        |   # first, check whether the corner is too low to the ground that the bottom homing will hit the ground (z < -400)
        |   lc_height = get_lift_column_height_condensed()
        |   # total height = zeroed lift column height (41.25 inches) (1.04775 m) plus lift column height plus robot relative height
        |   totalheight = 1.04775 + lc_height + point0[2]
        |   if totalheight < 1.04775 - 0.400:
        |     # bad
        |     popuptext = "Tank Corner is too low to the ground. Collisions will occur. Stop Program and raise tank. "
        |     # infinite loop
        |     while 1==1:
        |       popup(popuptext, title="Robot Positioning Warning",blocking=True)
        |     end
        |   end
        | 
        | 
        | 
        |   # next, check whether the touchpoints are reachable
        |   allvalid = check_structofpoints_validity(struct_touchpoints)
        |   if not allvalid:
        | 
        |     # then unreachable
        |     # generate message
        |     listproblems = ""
        |     listnames = ["ph1", "ph2", "ph3", "ph4", "ph5", "ph6", "ph7", "ph2up", "ph4up"]
        |     i = 0
        |     structlength = 9
        |     while i < structlength:
        |       curr = struct_touchpoints[i]
        |       valid = get_inverse_kin_has_solution(curr)
        |       if not valid:
        |         listproblems = listproblems + listnames[i]
        |       end
        |       i = i + 1
        |     end
        |     # display
        |     popuptext = "Robot is too far from tank corner. Cannot reach some necessary positions. Stop Program and move robot closer. " + listproblems
        |     # infinite loop
        |     while 1==1:
        |       popup(popuptext, title="Robot Positioning Warning",blocking=True)
        |     end
        |   end
        | 
        | end
        | 
        | # this function takes a struct of points as an argument, and checks whether every point in the list is reachable using get_inverse_kin_has_solution()
        | # this function does NOT check for weird twists or joint limits
        | # inputstruct must contain only points
        | # it returns true if all points are valid. it returns false if any points are valid
        | # a list of length 0 indicates that all points are valid
        | def check_structofpoints_validity(inputstruct):
        |   # next, check whether the touchpoints are reachable
        |   structlength = length(inputstruct)
        |   i = 0
        |   allvalid = True
        |   while i < structlength:
        |     curr = inputstruct[i]
        |     valid = get_inverse_kin_has_solution(curr)
        |     if not valid:
        |       return False
        |     end
        |     i = i + 1
        |   end
        |   return True
        | end
        | 
        | # checks the validity of all points during a left weld
        | # takes 2 arguments: struct1 (struct1[0] has to contain pointintersect) and struct2 (contains all the points (9) of the weld path)
        | def check_validity_left(struct1, struct2):
        |   #first, check whether robot is too close
        |   pointintersect = struct1[0]
        |   # next, check if the corner is too close to the robot to do a left around weld (complex but approximately X > -1300)
        |   # if y < 0, then x < -1300. if y < 480, then y > (1300+x)*8. if y > 480, then y > (1235+x)*4 + 500
        |   toocloseleftweld = False
        |   if pointintersect[1] < 0:
        |     if pointintersect[0] > -1.300:
        |       toocloseleftweld = True
        |     end
        |   elif pointintersect[1] < 0.480:
        |     if pointintersect[1] < (1.300 + pointintersect[0])*8:
        |       toocloseleftweld = True
        |     end
        |   else:
        |     if pointintersect[1] < (1.235 + pointintersect[0])*4 + 0.500:
        |       toocloseleftweld = True
        |     end
        |   end
        |   if toocloseleftweld:
        |     # bad
        |     popuptext = "Robot is too close to tank corner. Collisions may occur. Stop Program and move robot farther. "
        |     # infinite loop
        |     while 1==1:
        |       popup(popuptext, title="Robot Positioning Warning",blocking=True)
        |     end
        |   end
        | 
        |   #next, check whether all the points in the weldpath are valid
        |   structlength = 9
        |   i = 0
        |   allvalid = True
        |   listproblems = ""
        |   listnames = ["point1", "point2", "point4", "point5", "point_1", "point_2", "point_3", "point_4", "point_5"]
        |   while i < structlength:
        |     curr = struct2[i]
        |     valid = get_inverse_kin_has_solution(curr)
        |     if not valid:
        |       allvalid = False
        |       listproblems = listproblems + listnames[i]
        |     end
        |     i = i + 1
        |   end
        | 
        |   if not allvalid:
        |     # display
        |     popuptext = "Robot is too far from tank corner. Cannot reach some necessary positions. Stop Program and move robot closer. " + listproblems
        |     # infinite loop
        |     while 1==1:
        |       popup(popuptext, title="Robot Positioning Warning",blocking=True)
        |     end
        |   end
        | 
        |   # check whether the path involves weird turns or joint limits. currently just checks the first position
        |   p_prev = [-0.021118, -1.26292, 2.43578, 5.07088, -2.29912, 1.53362] #last point of left weld prerotate
        |   joints_1 = get_inverse_kin(struct2[0], p_prev) # struct2[0] is point1
        |   allGood = True
        |   i = 0
        |   structlength = 6
        |   while i < structlength:
        |     joint_curr = joints_1[i]
        |     # check for anything that exceeds joint limits
        |     degreesmax = 360 * pi / 180
        |     if joint_curr > degreesmax or joint_curr < degreesmax * -1:
        |       allGood = False
        |     end
        |     # check for anything that is significantly different than the aligned approach. could indicate a twist is needed. we dont want that
        |     maxdifference = 150 * pi / 180
        |     difference = joint_curr - p_prev[i]
        |     if difference > maxdifference or difference * -1 > maxdifference:
        |       allGood = False
        |     end
        |     i = i + 1
        |   end
        | 
        |   if not allGood:
        |     # call lift column extend function
        |     struct2 = floor_corner_lift_column_extend_left(struct2)
        | 
        |   end
        | 
        |   # return struct2 back
        |   return struct2
        | end
        | 
        | # checks the validity of all points during a right weld
        | def check_validity_right(struct1, struct2):
        |   # first, check whether the right pivot will bonk itself
        |   pointintersect = struct1[0]
        |   heading1 = struct1[1] # this is the direction that the welder will face when doing the right side of the box
        | 
        |   #first, check whether the heading is just too far offset
        |   # more than 15 degrees off of 45 is too much
        |   # normal heading is 216 degrees
        |   #201 degrees to 231 degrees
        |   heading1degrees = heading1 * 180 / pi
        |   if heading1degrees < 201 or heading1degrees > 231 :
        |     # then out of range
        |     popuptext = "Robot is not aligned at a 45 degree angle of corner (15 degree leeway). Collisions may occur. Stop Program and align robot. heading1degrees=" + str_cat("",heading1degrees)
        |     # infinite loop
        |     while 1==1:
        |       popup(popuptext, title="Robot Positioning Warning",blocking=True)
        |     end
        |   end
        | 
        |   #TODO: add the checks for whether x is too close, given the heading
        |   # add checks for whether x is too close, given the heading
        |   # different equations for whether heading offset > 5 degrees or less (inc. negative)
        |   headingoffset = heading1degrees - 216
        |   if headingoffset < 5:
        |     # then calculate a and b
        |     a = 0.4584 + -0.02369 * headingoffset
        |     b = (-1151.4 + 13.83 * headingoffset) / 1000
        |     # check whether x > a*y+b
        |     if pointintersect[0] > a * pointintersect[1] + b:
        |       # bad
        |       popuptext = "Robot is too close to tank corner or not at the right angle. Collisions may occur. Stop Program and align robot. "
        |       # infinite loop
        |       while 1==1:
        |         popup(popuptext, title="Robot Positioning Warning",blocking=True)
        |       end
        |     end
        |   else:
        |     # headingoffset > 5 degrees
        |     if pointintersect[1] < 0:
        |       if pointintersect[0] > -1150.0 / 1000.0:
        |         #bad
        |         popuptext = "Robot is too close to tank corner. Collisions may occur. Stop Program and align robot. "
        |         # infinite loop
        |         while 1==1:
        |           popup(popuptext, title="Robot Positioning Warning",blocking=True)
        |         end
        |       end
        |     else:
        |       # if x > .7736 y - 1101.9 then bad
        |       if pointintersect[0] > 0.7736 * pointintersect[1] - 1101.9 / 1000:
        |         popuptext = "Robot is too close to tank corner. Collisions may occur. Stop Program and align robot. "
        |         # infinite loop
        |         while 1==1:
        |           popup(popuptext, title="Robot Positioning Warning",blocking=True)
        |         end
        |       end
        |     end
        |   end
        | 
        |   #next, check whether all the points in the weldpath are valid
        |   structlength = 9
        |   i = 0
        |   allvalid = True
        |   listproblems = ""
        |   listnames = ["point1", "point2", "point4", "point5", "point_1", "point_2", "point_3", "point_4", "point_5"]
        |   while i < structlength:
        |     curr = struct2[i]
        |     valid = get_inverse_kin_has_solution(curr)
        |     if not valid:
        |       allvalid = False
        |       listproblems = listproblems + listnames[i]
        |     end
        |     i = i + 1
        |   end
        | 
        |   if not allvalid:
        |     # display
        |     popuptext = "Robot is too far from tank corner. Cannot reach some necessary positions. Stop Program and move robot closer. " + listproblems
        |     # infinite loop
        |     while 1==1:
        |       popup(popuptext, title="Robot Positioning Warning",blocking=True)
        |     end
        |   end
        | 
        |   # check whether the path involves weird turns or joint limits. currently just checks the first position
        |   p_prev = [-1.13307, -1.48911, 2.84785, 4.92357, -4.89059, 1.57184] #last point of right weld prerotate
        |   joints_1 = get_inverse_kin(struct2[0], p_prev) # struct2[0] is point1
        |   allGood = True
        |   i = 0
        |   structlength = 6
        |   while i < structlength:
        |     joint_curr = joints_1[i]
        |     # check for anything that exceeds joint limits
        |     degreesmax = 360 * pi / 180
        |     if joint_curr > degreesmax or joint_curr < degreesmax * -1:
        |       allGood = False
        |     end
        |     # check for anything that is significantly different than the aligned approach. could indicate a twist is needed. we dont want that
        |     maxdifference = 150 * pi / 180
        |     difference = joint_curr - p_prev[i]
        |     if difference > maxdifference or difference * -1 > maxdifference:
        |       allGood = False
        |     end
        |     i = i + 1
        |   end
        | 
        |   if not allGood:
        |     struct2 = floor_corner_lift_column_extend_right(struct2)
        |   end
        | 
        |   # return struct2 back
        |   return struct2
        | end
        | 
        | def floor_corner_lift_column_extend_right(struct2):
        |   # we know that p1 cannot be accessed without a twist
        |   # calculate the height needed to get to p1
        |   liftcolumnincrement = 2.0 # mm
        |   enoughHeightAdded = False
        |   liftColumnHeightTest = 0
        |   while not enoughHeightAdded:
        |     liftColumnHeightTest = liftColumnHeightTest + liftcolumnincrement
        |     # set the orig_joints for p1. p1 demo was joint angles of [-0.45, -31.79, 56.47, 333.06, -130.98, 87.87] (degrees)
        |     # which equals [-0.007853981633974475, -0.5548401692089968, 0.985587428601197, 5.812993606692308, -2.28603225426217, 1.5336208137274159]
        |     orig_joints = [-0.007853981633974475, -0.5548401692089968, 0.985587428601197, 5.812993606692308, -2.28603225426217, 1.5336208137274159]
        |     # get the modified point:
        |     origp1 = struct2[0]
        |     testp1 = p[origp1[0], origp1[1], origp1[2] - liftColumnHeightTest / 1000.0, origp1[3], origp1[4], origp1[5]]
        |     testpa1 = p[origp1[0]+0.05, origp1[1]+0.05, origp1[2] - liftColumnHeightTest / 1000, origp1[3], origp1[4], origp1[5]]
        |     enoughHeightAdded = can_pose_be_reached_without_twist(testp1, orig_joints) and can_pose_be_reached_without_twist(testpa1, orig_joints)
        |   end
        | 
        |   origp2 = struct2[1]
        |   testp2 = p[origp2[0], origp2[1], origp2[2] - liftColumnHeightTest / 1000.0, origp2[3], origp2[4], origp2[5]]
        |   origp4 = struct2[2]
        |   testp4 = p[origp4[0], origp4[1], origp4[2] - liftColumnHeightTest / 1000, origp4[3], origp4[4], origp4[5]]
        |   origp5 = struct2[3]
        |   testp5 = p[origp5[0], origp5[1], origp5[2] - liftColumnHeightTest / 1000, origp5[3], origp5[4], origp5[5]]
        | 
        | 
        | 
        |   liftcolumnzneeded = liftColumnHeightTest
        |   ret = struct(point1=testp1,point2=testp2,point4=testp4,point5=testp5,point_1=struct2[4],point_2=struct2[5],point_3=struct2[6],point_4=struct2[7],point_5=struct2[8])
        |   return ret
        | 
        | end
        | 
        | # this function gets called if you are doing a left floor corner extended, and the top is too high to reach (twists, etc.)
        | # this function takes the struct2 of weld points and modifies them (by subtracting from z) until the first weld point is reachable.
        | # it determines the height that the lift column needs to raise to make the first point reachable
        | # it then checks whether that height will allow the other points to be reachable
        | # if its all good, it sets the global variable liftcolumnzneeded, modifies struct2's points, and returns struct2
        | # if its not all good, then it displays an error message popup.
        | def floor_corner_lift_column_extend_left(struct2):
        |   # we know that p1 cannot be accessed without a twist
        |   # calculate the height needed to get to p1
        |   liftcolumnincrement = 2 # mm
        |   enoughHeightAdded = False
        |   liftColumnHeightTest = 0
        |   while not enoughHeightAdded:
        |     liftColumnHeightTest = liftColumnHeightTest + liftcolumnincrement
        |     # set the orig_joints for p1. p1 demo was joint angles of [-0.45, -31.79, 56.47, 333.06, -130.98, 87.87] (degrees)
        |     # which equals [-0.007853981633974475, -0.5548401692089968, 0.985587428601197, 5.812993606692308, -2.28603225426217, 1.5336208137274159]
        |     orig_joints = [-0.007853981633974475, -0.5548401692089968, 0.985587428601197, 5.812993606692308, -2.28603225426217, 1.5336208137274159]
        |     # get the modified point:
        |     origp1 = struct2[0]
        |     testp1 = p[origp1[0], origp1[1], origp1[2] - liftColumnHeightTest / 1000, origp1[3], origp1[4], origp1[5]]
        |     enoughHeightAdded = can_pose_be_reached_without_twist(testp1, orig_joints)
        |   end
        | 
        |   # check whether the other 3 points are valid
        |   valid = True
        |   # get the modified point
        |   origp2 = struct2[1]
        |   testp2 = p[origp2[0], origp2[1], origp2[2] - liftColumnHeightTest / 1000, origp2[3], origp2[4], origp2[5]]
        |   # p2 demo was joint angles of [-0.45, -21.2, 56.98, 321.95, -130.97, 87.85] (degrees)
        |   # which equals [-0.007853981633974475, -0.3700098014227975, 0.9944886077863679, 5.619087526795738, -2.285857721336971, 1.5332717478770168]
        |   orig_joints = [-0.007853981633974475, -0.3700098014227975, 0.9944886077863679, 5.619087526795738, -2.285857721336971, 1.5332717478770168]
        |   valid = valid and can_pose_be_reached_without_twist(testp2, orig_joints)
        |   # get the modified point
        |   origp4 = struct2[2]
        |   testp4 = p[origp4[0], origp4[1], origp4[2] - liftColumnHeightTest / 1000, origp4[3], origp4[4], origp4[5]]
        |   # p4 demo was joint angles of [-8.62, -43.23, 99.53, 213.86, -89.19, 40.78] (degrees)
        |   # which equals [-0.15044738152191103, -0.7545058356371478, 1.7371262045099545, 3.7325611383150696, -1.556659159853741, 0.7117452689632868]
        |   orig_joints = [-0.15044738152191103, -0.7545058356371478, 1.7371262045099545, 3.7325611383150696, -1.556659159853741, 0.7117452689632868]
        |   valid = valid and can_pose_be_reached_without_twist(testp4, orig_joints)
        |   # get the modified point
        |   origp5 = struct2[3]
        |   testp5 = p[origp5[0], origp5[1], origp5[2] - liftColumnHeightTest / 1000, origp5[3], origp5[4], origp5[5]]
        |   # p5 demo was joint angles of [-0.59, -34.36, 77.71, 226.7, -89.18, 48.81] (degrees)
        |   # which equals [-0.010297442586766533, -0.5996951309852511, 1.356295361724792, 3.9566614142711405, -1.5564846269285415, 0.8518952078984314]
        |   orig_joints = [-0.010297442586766533, -0.5996951309852511, 1.356295361724792, 3.9566614142711405, -1.5564846269285415, 0.8518952078984314]
        |   valid = valid and can_pose_be_reached_without_twist(testp5, orig_joints)
        | 
        |   if not valid:
        |     # display
        |     popuptext = "Top of Weld is too high above robot. Cannot reach some necessary positions. Stop Program and try again with a lower top point. "
        |     # infinite loop
        |     while 1==1:
        |       popup(popuptext, title="Robot Positioning Warning",blocking=True)
        |     end
        |   else:
        |     liftcolumnzneeded = liftColumnHeightTest
        |     ret = struct(point1=testp1,point2=testp2,point4=testp4,point5=testp5,point_1=struct2[4],point_2=struct2[5],point_3=struct2[6],point_4=struct2[7],point_5=struct2[8])
        |     return ret
        |   end
        | end
        | 
        | # this function calculates whether a given pose can be reached, and if it can, whether it requires a wrist twist (from the seed joint angles)
        | # arguments are target pose (p[x,y,z,rx,ry,rz]) and orig_joints which is the 6 joint angles of a pose that is close by the target pose and has the desired joint angles
        | # returns true if the pose is valid and requires no twist. If pose is valid but requires a twist, returns false. If pose is invalid, returns false.
        | def can_pose_be_reached_without_twist(pose, orig_joints):
        |   # first, determine if the pose is valid
        |   valid = get_inverse_kin_has_solution(pose)
        |   if not valid:
        |     return False
        |   end
        |   joints_1 = get_inverse_kin(pose, orig_joints)
        |   #iterate through the 6 joints
        |   allGood = True
        |   i = 0
        |   structlength = 6
        |   while i < structlength:
        |     joint_curr = joints_1[i]
        |     # check for anything that exceeds joint limits
        |     degreesmax = 360 * pi / 180
        |     if joint_curr > degreesmax or joint_curr < degreesmax * -1:
        |       allGood = False
        |     end
        |     # check for anything that is significantly different than the aligned approach. could indicate a twist is needed. we dont want that
        |     maxdifference = 150 * pi / 180
        |     difference = joint_curr - orig_joints[i]
        |     if difference > maxdifference or difference * -1 > maxdifference:
        |       allGood = False
        |     end
        |     i = i + 1
        |   end
        |   return allGood
        | end
        | 
        | # this function sends a signal to turn extrusion on
        | def turn_extrusion_on():
        |   # flush the channel
        |   resp0 = send_serial_signal(["u", "r", "?"])
        |   # send the signal
        |   resp1 = send_serial_signal(["u", "R", "1"])
        |   # if resp <> "uR1"
        |   if resp1 != [252,82,49]:
        |     # turn off extrusion and heating. inform calvin
        |     resp2 = send_serial_signal(["u", "R", "0"])
        |     resp3 = send_serial_signal(["u", "H", "0"])
        |     popuptext = "Error code encountered while trying to start extrusion. Find Calvin. "
        |     while 1==1:
        |       popup(popuptext, title="Extrusion Error Code",blocking=True)
        |       popup(resp1, blocking=True)
        |     end
        |   end
        | end
        | 
        | # this function sends a signal and receives a response
        | # signal is a list of 3 strings, 1 character each. first is u. second is the next character. third is final character
        | def send_serial_signal(signal):
        |   signal2char = signal[1]
        |   signal3char = signal[2]
        |   listsignal = [252, get_corr_number(signal2char), get_corr_number(signal3char)]
        |   resp1 = WTSerialBridge.send_command("/dev/ttyUSB0",1200, 8, "None", "One", "None", 1000, "None", "None", listsignal, True)
        |   return resp1
        | end
        | 
        | # this function converts a letter into its ascii number
        | def get_corr_number(letter):
        |   if letter == "A":
        |     return 65
        |   elif letter == "H":
        |     return 72
        |   elif letter == "R":
        |     return 82
        |   elif letter == "M":
        |     return 77
        |   elif letter == "E":
        |     return 69
        |   elif letter == "a":
        |     return 97
        |   elif letter == "b":
        |     return 98
        |   elif letter == "h":
        |     return 104
        |   elif letter == "r":
        |     return 114
        |   elif letter == "s":
        |     return 115
        |   elif letter == "m":
        |     return 109
        |   elif letter == "0":
        |     return 48
        |   elif letter == "1":
        |     return 49
        |   elif letter == "2":
        |     return 50
        |   elif letter == "3":
        |     return 51
        |   elif letter == "4":
        |     return 52
        |   elif letter == "5":
        |     return 53
        |   elif letter == "6":
        |     return 54
        |   elif letter == "7":
        |     return 55
        |   elif letter == "8":
        |     return 56
        |   elif letter == "9":
        |     return 57
        |   elif letter == "?":
        |     return 63
        |   end
        | end
        | 
        | # this function checks whether the welder is in the ready state.
        | # to be called at the beginning of Main Program
        | def welder_state_ready():
        |   # flush the channel
        |   resp0 = send_serial_signal(["u", "s", "?"])
        |   # send the signal
        |   resp1 = send_serial_signal(["u", "s", "?"])
        |   # if resp1 == [252,115,49] (us1) then it is ready. otherwise, it is not
        |   if resp1 != [252,115,49]:
        |     popuptext = "Welder is not ready for extrusion. Follow the instructions to start heating welder. "
        |     while 1==1:
        |       popup(popuptext, title="Welder Not Ready",blocking=True)
        |     end
        |   end
        | 
        | end
        | 
        | def get_lift_column_height():
        |   # begin: URCap Program Node
        |   #   Source: MachineLogic for Universal Robots, 3.1.7, Vention Inc.
        |   #   Type: MachineLogic for Universal Robots
        |   #$ 5 "MachineLogic Get Position"
        |   while isVentionMovementBusyMachineMotion1==True:
        |     sleep(0.05)
        |   end
        |   if(isVentionMovementBusyMachineMotion1 == False):
        |     isVentionMovementBusyMachineMotion1 = True
        |     socket_send_string("estop/status;", "MachineMotion1")
        |     temp_estop_var_vention = socket_read_string("MachineMotion1",timeout=15)
        |     while(temp_estop_var_vention=="estop/status true"):
        |       if temp_estop_var_vention=="estop/status true":
        |         sendStringWithTimeout("estop/systemreset/request","Ack estop/systemreset/request;","MachineMotion1")
        |       end
        |       socket_send_string("estop/status;", "MachineMotion1")
        |       temp_estop_var_vention = socket_read_string("MachineMotion1",timeout=15)
        |       if temp_estop_var_vention=="estop/status true":
        |         popup("MachineMotion in estop, make sure you have all emergency modules released manually. If you continue the system will try to reset MachineMotion automatically.",blocking=True)
        |       end
        |     end
        |   else:
        |     popup("resource is being used already: MachineMotion1")
        |     halt
        |   end
        |   socket_send_string("GET im_get_controller_pos_axis_1;", "MachineMotion1")
        |   temp_drive = socket_read_ascii_float(1, "MachineMotion1",timeout=15)
        |   global var_1 = temp_drive[1]
        |   isVentionMovementBusyMachineMotion1 = False
        |   sleep(0.03)
        |   # end: URCap Program Node
        | end
        | 
        | def get_lift_column_height_condensed():
        |   socket_send_string("GET im_get_controller_pos_axis_1;", "MachineMotion1")
        |   temp_drive = socket_read_ascii_float(1, "MachineMotion1",timeout=15)
        |   ret = temp_drive[1]
        |   return ret
        | end
  'list possible points'
  Folder robot 1 moves
    If 1≟2
      MoveJ speed 60 deg/s, acceleration 80 deg/s^2 (useActiveTCP=true optimoveEnabled=false optiMoveSpeed=0.3 optiMoveAcceleration=0.09) feature=Base
        Waypoint r1_ek_oldhome: TCP in base x=397.38 y=356.254 z=319.821 mm, rx=2.3163 ry=2.0576 rz=0.0741 rad; joints [-198.126, -117.851, 133.303, -13.009, -11.422, -6.035] deg; TCP offset x=-5.49 y=-328 z=106.39 mm, rx=1.2092 ry=-1.2092 rz=1.2092 rad
        Waypoint r1_ek_extrude: TCP in base x=454.852 y=405.449 z=64.015 mm, rx=2.3168 ry=2.0514 rz=0.0767 rad; joints [-187.624, -89.406, 141.395, -19.732, -0.818, -36.116] deg
        Waypoint r1_ek_front: TCP in base x=439.065 y=405.452 z=65.996 mm, rx=2.3168 ry=2.0514 rz=0.0766 rad; joints [-187.962, -93.321, 143.386, -27.168, -1.131, -26.752] deg
        Waypoint r1_ek_middle: TCP in base x=419.01 y=404.851 z=65.995 mm, rx=2.3096 ry=2.0447 rz=0.0891 rad; joints [-188.553, -97.485, 146.002, -33.769, -1.69, -19.324] deg
        Waypoint r1_ek_middle2: TCP in base x=417.012 y=405.435 z=65.003 mm, rx=2.3169 ry=2.0513 rz=0.0766 rad; joints [-188.493, -97.025, 145.794, -33.21, -1.638, -19.415] deg
        Waypoint r1_ek_bottom: TCP in base x=413.072 y=405.431 z=68 mm, rx=2.3168 ry=2.0513 rz=0.0767 rad; joints [-188.596, -97.887, 146.02, -33.517, -1.738, -18.475] deg
        Waypoint r1_ek_end: TCP in base x=389.999 y=405.444 z=68.005 mm, rx=2.3169 ry=2.0514 rz=0.0766 rad; joints [-189.248, -101.07, 148.002, -36.337, -2.38, -14.447] deg
  Folder robot 2 moves
    If 1≟2
      MoveJ speed 60 deg/s, acceleration 80 deg/s^2 (useActiveTCP=true optimoveEnabled=false optiMoveSpeed=0.3 optiMoveAcceleration=0.09) feature=Base
        Waypoint r2_ek_oldhome: TCP in base x=397.38 y=356.254 z=319.821 mm, rx=2.3163 ry=2.0576 rz=0.0741 rad; joints [-198.308, -118.162, 133.451, -12.562, -11.515, -6.325] deg; TCP offset x=-9.5 y=-328 z=105.73 mm, rx=1.2092 ry=-1.2092 rz=1.2092 rad
        SuppressedNode
          Waypoint Waypoint_1: TCP in base x=612.886 y=429.305 z=100.477 mm, rx=1.8619 ry=2.4807 rz=0.0957 rad; joints [-182.793, -81.736, 125.569, -42.478, -18.966, -5.44] deg
        Waypoint r2_ek_extrude: TCP in base x=612.886 y=429.305 z=100.477 mm, rx=2.15 ry=2.2258 rz=0.0874 rad; joints [-183.316, -85.158, 129.692, -39.696, -5.262, -8.969] deg
        Waypoint r2_ek_front: TCP in base x=556.405 y=429.305 z=76.984 mm, rx=-2.1704 ry=-2.2682 rz=-0.0159 rad; joints [-183.513, -85.623, 132.794, -41.666, -5.994, -5.809] deg
        Waypoint r2_ek_middle: TCP in base x=550.034 y=429.305 z=76.254 mm, rx=-2.1704 ry=-2.2682 rz=-0.0159 rad; joints [-183.554, -85.983, 133.283, -41.831, -6.035, -5.773] deg
        Waypoint r2_ek_bottom: TCP in base x=546.595 y=429.305 z=80.868 mm, rx=-2.1704 ry=-2.2682 rz=-0.0159 rad; joints [-183.576, -86.513, 133.34, -41.373, -6.058, -5.758] deg
        Waypoint r2_ek_end: TCP in base x=537.335 y=429.305 z=80.868 mm, rx=-2.1704 ry=-2.2682 rz=-0.0159 rad; joints [-183.639, -87.118, 134.001, -41.482, -6.12, -5.705] deg
  'detemine correct points for which robot'
  If robot_number≟1
    Folder robot1 positions
      ek_oldhome := r1_ek_oldhome_p
      ek_extrude := r1_ek_extrude_p
      ek_front := r1_ek_front_p
      ek_middle := r1_ek_middle_p
      ek_middle2 := r1_ek_middle2_p
      ek_bottom := r1_ek_bottom_p
      ek_end := r1_ek_end_q
  ElseIf robot_number≟2
    Folder robot1 positions
      ek_oldhome := r2_ek_oldhome_p
      ek_extrude := r2_ek_extrude_p
      ek_front := r2_ek_front_p
      ek_middle := r2_ek_middle_p
      ek_middle2 := r2_ek_middle_p
      ek_bottom := r2_ek_bottom_p
      ek_end := r2_ek_end_q
  'start of program'
  SuppressedNode
    SafeHome (positionOptionType=SPEED_AND_ACCELERATION speed=1.047198 acceleration=1.396263 nextMotionTime=2)
  Set NoAction tcp=pretend_welder
  MoveJ speed 60 deg/s, acceleration 80 deg/s^2 (useActiveTCP=true optimoveEnabled=false optiMoveSpeed=0.3 optiMoveAcceleration=0.09) feature=Base
    SuppressedNode
      Waypoint r1_ek_oldhome: TCP in base x=397.38 y=356.254 z=319.821 mm, rx=2.3163 ry=2.0576 rz=0.0741 rad; joints [-198.126, -117.851, 133.303, -13.009, -11.422, -6.035] deg; TCP offset x=-5.49 y=-328 z=106.39 mm, rx=1.2092 ry=-1.2092 rz=1.2092 rad
    Waypoint Variable (Variable): variable=ek_oldhome
    'above waypoint is home'
  'move above bucket'
  MoveJ speed 60 deg/s, acceleration 80 deg/s^2 (useActiveTCP=true optimoveEnabled=false optiMoveSpeed=0.3 optiMoveAcceleration=0.09) feature=Base
    SuppressedNode
      Waypoint r1_ek_extrude: TCP in base x=454.852 y=405.449 z=64.015 mm, rx=2.3168 ry=2.0514 rz=0.0767 rad; joints [-187.624, -89.406, 141.395, -19.732, -0.818, -36.116] deg
    Waypoint Variable (Variable): variable=ek_extrude
  'extrude out a foot'
  SuppressedNode
    Script: turn_extrusion_on()
  URCap WireTank Serial (WireTank Serial, WireTank, LLC) dataModel(NODE_TITLE=Serial Bridge uR1, Command=[252,82,49], QUERY=false, OUTPUT_ENTRY=Static, byte_array=true, Variable(key=OUTPUT_VARIABLE, variable=HwResp))
  Set DigitalOutput pin=digital_out[0]; digitalValue=1
  Wait Sleep waitTime=24
  SuppressedNode
    Wait Sleep waitTime=2
  URCap WireTank Serial (WireTank Serial, WireTank, LLC) dataModel(QUERY=false, NODE_TITLE=Serial Bridge uR0, Command=[252,82,48], byte_array=true, OUTPUT_ENTRY=Static, Variable(key=OUTPUT_VARIABLE, variable=HwResp))
  Wait Sleep waitTime=1
  Set DigitalOutput pin=digital_out[0]; digitalValue=0
  'slice'
  MoveL speed 30 mm/s, acceleration 50 mm/s^2 (useActiveTCP=true optimoveEnabled=false optiMoveSpeed=0.3 optiMoveAcceleration=0.09) feature=Base
    SuppressedNode
      Waypoint r1_ek_front: TCP in base x=439.065 y=405.452 z=65.996 mm, rx=2.3168 ry=2.0514 rz=0.0766 rad; joints [-187.962, -93.321, 143.386, -27.168, -1.131, -26.752] deg
    SuppressedNode
      Waypoint r1_ek_middle: TCP in base x=419.01 y=404.851 z=65.995 mm, rx=2.3096 ry=2.0447 rz=0.0891 rad; joints [-188.553, -97.485, 146.002, -33.769, -1.69, -19.324] deg
    SuppressedNode
      Waypoint r1_ek_middle2: TCP in base x=417.012 y=405.435 z=65.003 mm, rx=2.3169 ry=2.0513 rz=0.0766 rad; joints [-188.493, -97.025, 145.794, -33.21, -1.638, -19.415] deg
    SuppressedNode
      Waypoint r1_ek_bottom: TCP in base x=413.072 y=405.431 z=68 mm, rx=2.3168 ry=2.0513 rz=0.0767 rad; joints [-188.596, -97.887, 146.02, -33.517, -1.738, -18.475] deg
    SuppressedNode
      Waypoint r1_ek_end: TCP in base x=389.999 y=405.444 z=68.005 mm, rx=2.3169 ry=2.0514 rz=0.0766 rad; joints [-189.248, -101.07, 148.002, -36.337, -2.38, -14.447] deg
    Waypoint Variable (Variable): variable=ek_front
    Waypoint Variable (Variable): variable=ek_middle
    Waypoint Variable (Variable): variable=ek_middle2
    Waypoint Variable (Variable): variable=ek_bottom
    Waypoint Variable (Variable): variable=ek_end
  MoveJ speed 60 deg/s, acceleration 80 deg/s^2 (useActiveTCP=true optimoveEnabled=false optiMoveSpeed=0.3 optiMoveAcceleration=0.09) feature=Base
    SuppressedNode
      Waypoint r1_ek_oldhome: TCP in base x=397.38 y=356.254 z=319.821 mm, rx=2.3163 ry=2.0576 rz=0.0741 rad; joints [-198.126, -117.851, 133.303, -13.009, -11.422, -6.035] deg
    Waypoint Variable (Variable): variable=ek_oldhome
    'above waypoint is home'
  SuppressedNode
    SafeHome (positionOptionType=SPEED_AND_ACCELERATION speed=1.047198 acceleration=1.396263 nextMotionTime=2)
Thread Thread_1 (runOnlyOnce=true)
  Loop While (checkContinuously=false) expression=True
    If freedrive_m_var≟ True
      Script: freedrive_mode()
      free_dr_already := True
    Else 
      If free_dr_already
        Script: end_freedrive_mode()
    Script: sync()
SuppressedNode
  Thread Thread_2 (runOnlyOnce=false)
    Loop While (checkContinuously=false) expression=True
      If thread2trigger≟ True
        'do the dot extrude'
        Wait Sleep waitTime=5
        URCap WireTank Serial (WireTank Serial, WireTank, LLC) dataModel(byte_array=true, NODE_TITLE=Serial Bridge uR1, Command=[252,82,49], QUERY=false, OUTPUT_ENTRY=Static, Variable(key=OUTPUT_VARIABLE, variable(name=HwResp)))
        Wait Sleep waitTime=2
        URCap WireTank Serial (WireTank Serial, WireTank, LLC) dataModel(QUERY=false, NODE_TITLE=Serial Bridge uR0, Command=[252,82,48], byte_array=true, OUTPUT_ENTRY=Static, Variable(key=OUTPUT_VARIABLE, variable(name=HwResp)))
        thread2trigger := False
      Script: sync()
